FUNCTION_BLOCK Process EXTENDS BaseProcess
VAR_INPUT
END_VAR
VAR_OUTPUT
END_VAR
VAR_IN_OUT
END_VAR
VAR
	///At least 1 variable needed because subclass members of an empty class are not exposed by OPC UA (TwinCAT bug!)
	{attribute 'OPC.UA.DA' := '0'}
	testVar: BOOL;
END_VAR

IF do_request THEN
    do_request_result := request();
    do_request := FALSE;
END_IF;
SUPER^();

{attribute 'TcRpcEnable' := '1'}
METHOD start
VAR_INPUT
END_VAR
VAR_OUTPUT
END_VAR
VAR_IN_OUT
END_VAR
VAR
END_VAR
THIS^.statuses.busyStatus( isBusy := TRUE );
THIS^.statuses.healthStatus( isGood := TRUE );
END_METHOD

{attribute 'TcRpcEnable' := '1'}
METHOD request : RequestResults
VAR_INPUT
END_VAR
VAR_OUTPUT
END_VAR
VAR_IN_OUT
END_VAR
VAR
END_VAR
IF THIS^.statuses.enabledStatus.enabled THEN
    THIS^.start();
    request := RequestResults.ACCEPTED;
ELSE
    request := RequestResults.REJECTED;
END_IF;
END_METHOD

END_FUNCTION_BLOCK

(* stored: Version 1.1.0.1, ProductVersion 3.1.4019.2
   POU Process: Id {6e61ff84-e51a-4a86-9866-54d9b302d1d8}, SpecialFunc None
   Method start: Id {001b4a03-7dc9-4f63-b7eb-2d1704b806df}
   Method request: Id {15d2ca4c-a902-4ee7-81ef-600adf7a289d} *)
